// TIA Portal V20 export
TYPE "LConSMC_typeTaperOutput"
// stored: Access Published
   STRUCT
      busy : Bool;   // TRUE: Der Funktionsbaustein ist aktiv / TRUE: The function block is active
      error : Bool := FALSE;   // TRUE: Es ist ein Fehler aufgetreten / TRUE: An error occured
      errorID : DWord := 16#0000_0000;   // Detaillierte Fehlerbeschreibung / Detailed error description
      tensionTaper : LReal := 1.0;   // Multiplikativer Wert der Zugabsenkung (0 - 1.0). Dieser Wert muss mit dem Zugsollwert multipliziert werden / Multiplicative value for tension reduction (0-1.0). The value must be multiplied with the tension setpoint
   END_STRUCT;
END_TYPE
